(* CODESYS project p7lib-basetypes.library
   Company: MacGregor
   DocFormat: reStructuredText
   DefaultNamespace: p7type
   Version: 1.2.7
   Placeholder: p7lib-basetypes
   Author: Ralph Koettlitz
   Title: p7lib-basetypes

Project tree, tasks and I/O mapping:
  AnalogOut/
    interface IAnalogOut: Value
  Common/
    interface IAMSADDR: AMSAddr
    interface IP6Identifier: ID, IDname
    interface IP6OpState: OpState
    interface IP6State: State
    data type P6IdName
    data type P6OpState
    data type P6State
  ControlUnits/
    data type ControlUnitStates
    interface IBaseControlUnit: ActionSignal, ActivateWinch, Alarm, AutoAvailable, AutoMode, Calibrate, CooperatingWinchIsRotating, Disable, InControl, IsInControlOf, JoystickInCentre, ManualTorqueRequested, ManualTorqueSignal, PotmeterRaw, PotmeterReference, ReleaseControl, RequestedWinchMode, SetSelectedWinch, StopWinch, TurtleMode, TurtleModeRequested, VelocityRaw, VelocityReference
    interface IFishpumpControl: Softstart, Speed, start, stop
    interface INethaulerControl: TiltIn, TiltOut
    interface ITrawlControlUnit: JoystickPORT, JoystickSTBD, PotentiometerPORT, PotentiometerSTBD, TDE, TensionMaster, TensionMaxRef, TorqueButtonPORT, TorqueButtonSTBD, VelocityMaster, VelocityMaxRef
  Electrical/
    Drive/
      data type ConfigDriveMux
      data type DriveCMD
      data type DriveGearSet
      data type DriveIInverterArray
      data type DriveIServiceArray
      data type DriveMuxAllocationData
      data type DriveMuxAllocationValue
      interface IDrive: getGearRatio, getInverterArray, getSpeed, getSpeedMax, getTorque, getTorqueMax, getTorqueRel, getTorqueRelMax, IDName, isActivationPossible, isAtZeroSpeed, OpState, setOperation, setProcessValues, State
      interface IDriveGearSet: setGearSet
      interface IDriveMux: acquire, areInvertersDeactivated, getActiveInverters, getAvailableInverters, getAverageMotorSpeed, getAverageTorqueRel, getInverter, getInverterInterface, getInvertersOwned, getMotorFactor, hasActiveInvertersMin, hasInvertersMin, isAllocationPossible, isAtZeroSpeed, isBusy, release, setInverterOperation, setMotors, setProcessValues, SplitMode, update, updateSpeedRef
    Inverter/
      interface IEncoder: changeDirectionRawValue, changeDirectionValue, DirectionValue, DirectionValueRaw, resetAll, Resolution, setValueTo, Value, ValueRaw
      interface IEncoderBlock: Length
      interface IInverter: AMSAddr, Event, EventId, getEncoder, getMotor, getOpTime, getPower, getSpeed, getTorqueRel, isAtZeroSpeed, OpState, resetOpTime, setMotor, setOperation, setProcessValues, State
      interface IMotor: Active, resetOpTime, Temperature
      data type InverterCMD
    PMS/
      data type AFE_CMD
      interface IAFE: ChargeOverload, Event, EventId, FieldbusProblem, getOpTime, ID, IDName, OpState, PassiveMode, Power, PowerRegen, setOperation, State
      interface IPMS: attachAFE, attachInverter, delAllAFE, delAllInverters, LimitPowerRegenUsage, LimitPowerUsage, PassiveMode, PowerRegenUsage, PowerUsage, StopPowerUsage
    Softstarter/
      interface ISoftstarter: Active, Enabled, Error, Local, OpTime, PowerUsage, Ready, reset, Running, start, stop
  EStop/
    interface IEmergencyStop: Activated, ActivatedSwitchIdx, ActivatedSwitchName
  Events/
    Alarm Class Definitions.txt
    Alarm Definitions.txt
    data type EventIdentifier
    data type UnitTypeID
  00000000-0000-0000-0000-000000000000|Events\Alarm Class Definitions.txt
  00000000-0000-0000-0000-000000000000|Events\Alarm Definitions.txt
  Hydraulics/
    HPU/
      interface IHPUBrake: Active, Error, PressureOK, setActive
    Valve/
      interface IValve: CalibrationMode, Error, setValve
      data type ValveCMD
  NtoMProtocol/
    interface IProtoBase1ToN: attach, getNoServices, getServiceByIdx, isAttached, resetService
    interface IProtoBaseNTo1: attach, getMasterByIdx, getNoMasters, isAttached, resetServices
    interface IProtocol
    interface IProtoMasterSingleService: attach, getService
    interface IProtoService
  PID/
    data type ConfigPID
    data type ConfigPID2P
    data type ConfigTrawlController
    interface IPID2DController: Error, Out, update
    interface IPIDController: Error, Out, update
  Sensor/
    interface IAnalogSensor: Error
    interface IAnalogSensorBase: Value, ValueRaw
  Winch/
    data type ClutchCMD
    data type ClutchStates
    data type FreeWheelingBrakeStates
    data type FreeWheelingBrakeUserCMD
    interface IAnchorWinch
    interface IBaseUserWinch: AssignControlUnitInControl, AutoMode, BoostAllowed, ControlCanBeReleased, getVelocityReference, ID, IsReadyToActivate, IsRotating, Length, ManMode, SafetyDistance, SetLengthNull, Speed, SpeedMax, State, Tension, Torque, TorqueMax, TorqueRel, Velocity, winchDriverStopped
    interface IClutch: ClutchState, ParkingBrakesOnWhileJoystickInCenterEnabled, SetClutchOperation
    interface IClutchAndBrake: BrakeOffPressure, BrakeOnPressure, ClutchState, FreeWheelingBrakeState, ParkingBrakesOnWhileJoystickInCenterEnabled, SetClutchOperation, SetFreeWheelingBrakeOperation
    interface IFishpump: DifferentialPressure, EnvironmentalPressure, MotorhousePressure, OilTemperature, PressureLow, TemperatureHigh
    interface INetHaulerWinch: TiltIn, TiltOut
    interface ISpool: confirmWirePosition, HeadPosition, Name, OpState, PIDError, setManualOperation, setOffsetDiamondScrew, setOperation, setSpoolEndPositionInner, setSpoolEndPositionOuter, Speed, State
    interface ITrawlModeController: HaulInModeAllowed, LengthDifference, LengthDifferenceMax, LengthDifferenceWarning, LengthMaster, LengthSetpoint, PayoutModeAllowed, SafetyLength, setOperation, setSounderDifferenceToZero, SnagControl, SounderLengthDifference, SounderLengthDifferenceMax, SounderLengthDifferenceWarning, TDE, TowingModeAllowed
    interface ITrawlWinch: AutoAvailable, AutoMode, Radius, SafetyDistance, setOperation, TorqueAuto, VelocityAuto
    interface IWinchMode: Mode
    data type ManualSpoolCMD
    data type SpoolCMD
    data type TrawlMaster
    data type TrawlWinchCMD
    data type UserWinchStates
    data type WinchAutoModes
    data type WinchManualModes
    data type WinchModes
  global variables CycleTimeConstants
  global variables Math
  global variables Parameters
*)

// Common/P6IdName
TYPE 
	P6IdName : STRING(32) := 'HAS NO NAME'; 
END_TYPE

// Common/P6OpState
{attribute 'qualified_only'}
{attribute 'strict'}
(*
State For Operations
====================

These values are giving an information whether a unit is running or not
*)
TYPE P6OpState :
(
	NOTAVAILABLE	:= -1,
	STOPPED			:= 0,
	PAUSING			:= 1,
	PREPARE			:= 2,
	RUN  			:= 3
);
END_TYPE

// Common/P6State
{attribute 'qualified_only'}
{attribute 'strict'}
(*
Device State
============

These states are similar to the Ethercat statemachine. Don't confuse these states with
states for operation
*)
TYPE P6State :
(
	BUSY 		:= -1,			// no access because of concurrent operation
	INIT 		:= 0,			// Initializing objects
	PREOP 		:= 1,			// Check whether operation is possible
	OP			:= 2			// Full operational
) INT;
END_TYPE

// ControlUnits/ControlUnitStates
// The different states a control unit can be in.
{attribute 'qualified_only'}
{attribute 'strict'}
TYPE ControlUnitStates :
(
	INIT 		:= 0,
	MONITORING 	:= 1,
	REQ_CONTROL := 2,
	IN_CONTROL 	:= 3,
	CALIBRATE 	:= 4,
	PAYOUT		:= 5,
	HAULIN		:= 6,
	TOW			:= 7
);
END_TYPE

// Electrical/Drive/ConfigDriveMux
TYPE ConfigDriveMux :
	STRUCT
		ID						: DINT				:= -666;
		name					: P6IdName			:= '';
		contextChangeTimeMax	: TIME 				:= T#5S;
		contextChangeTimeMin	: TIME				:= T#1S;
	END_STRUCT
END_TYPE

// Electrical/Drive/DriveCMD
{attribute 'qualified_only'}
{attribute 'strict'}
TYPE DriveCMD:
(
	NONE 		:= 0,
	ACTIVATE 	:= 1, 	// Go to run state, magnetized and no motor change. 
	PAUSE 		:= 2,
	STOP 		:= 3, 	// Stop motor connected to inverter.
	RESET 		:= 4, 	// Reset inverter faults.
	FASTSTOP	:= 5
) INT;
END_TYPE

// Electrical/Drive/DriveGearSet
{attribute 'qualified_only'}
{attribute 'strict'}
TYPE DriveGearSet :
(
	DEFAULT := 0,
	SET2	:= 1
) DINT;
END_TYPE

// Electrical/Drive/DriveIInverterArray
// Array for inverters per drive
TYPE DriveIInverterArray : ARRAY[0..Parameters.InverterPoolSize-1] OF IInverter; END_TYPE

// Electrical/Drive/DriveIServiceArray
// Muxer Inverter Array
TYPE DriveIServiceArray : ARRAY[0..Parameters.MuxerInverterPoolSize-1] OF IProtoService; END_TYPE

// Electrical/Drive/DriveMuxAllocationData
(*
This type is used to configure allocation priority values in ConfigInverter. 
*) 
TYPE 
	DriveMuxAllocationData : 
		ARRAY[0..Parameters.MuxerInverterPoolSize-1] OF DriveMuxAllocationValue := 
			[Parameters.MuxerInverterPoolSize(DriveMuxAllocationValue.LVL_NIL)]; 
END_TYPE

// Electrical/Drive/DriveMuxAllocationValue
{attribute 'qualified_only'}
TYPE DriveMuxAllocationValue :
(
	LVL_NIL 	:= -1,
	LVL_1		:= 0,
	LVL_2		:= 1,
	LVL_3		:= 2,
	LVL_4		:= 3,
	LVL_NO_SW	:= 100
) DINT;
END_TYPE

// Electrical/Inverter/InverterCMD
{attribute 'qualified_only'}
{attribute 'strict'}
TYPE InverterCMD:
(
	NONE 		:= 0,
	ACTIVATE 	:= 1, 	// Go to run state, magnetized and no motor change. 
	PAUSE 		:= 2,
	STOP 		:= 3, 	// Stop motor connected to inverter.
	RESET 		:= 4 	// Reset inverter faults.
) INT;
END_TYPE

// Electrical/PMS/AFE_CMD
{attribute 'qualified_only'}
{attribute 'strict'}
TYPE AFE_CMD:
(
	NONE 		:= 0,
	RUN			:= 1, 
	STOP 		:= 3, 	// Stop motor connected to inverter.
	RESET 		:= 4 	// Reset inverter faults.
) INT;
END_TYPE

// Events/EventIdentifier
{attribute 'qualified_only'}
{attribute 'strict'}
TYPE EventIdentifier :
	(	
		NO_ERROR 														:= 16#00000000,
		
		// Inverters
		INVERTER_NO_POWER_SUPPLY										:= 16#00000001, // No power supply for the motor
		INVERTER_OVERVOLTAGE 											:= 16#00000002, // Inverter is indicating too much voltage 
		INVERTER_TRIPPED 												:= 16#00000003, // Inverter is indicating error
		INVERTER_COMM_FAULT 											:= 16#00000004, // Fieldbus problem
		INVERTER_WRONG_MOTOR	 										:= 16#00000005,	// Invalid motor number
		INVERTER_LOCAL 													:= 16#00000006, // Inverter is in local mode
		INV_NO_READYREF		 											:= 16#00000007, // Inverter doesn't build magnet field 
		INVERTER_NO_CONTACTOR_MSG 										:= 16#00000008, // Contactor signal indicates wrong state
		INVERTER_RESET_REQUEST 											:= 16#00000009,		
		INVERTER_NO_DC													:= 16#0000000A, // Frontend doesn't deliver DC
		
		// Drives
		DRIVE_NOT_ENOUGH_MOTORS 										:= 16#00000010, // When the number of motors is too low
		DRIVE_ACTIVATION_FAILED 										:= 16#00000011, // When an inverter couldn't be activated.
		DRIVE_NO_ENCODERS_AVAILABLE										:= 16#00000012, // Encoder isn't working 
		DRIVE_DIRECT_ENCODER_CHOICE_WRONG								:= 16#00000013,	// config.Option_OnlyThisInverterHasEncoder >= NumberOfInvertersMax	 

		// Winch Base 
		WINCHBASE_AUTOMODE_LARGELAG										:= 16#00000020,	// Too large lag between setpoint and length
		WINCHBASE_DRIVE_IS_NOT_AVAILABLE								:= 16#00000021,
		WINCHBASE_SPOOL_IS_NOT_AVAILABLE								:= 16#00000022, // The drive for spooling is down
	 
		// Encoder
		ENCODER_COUNTER_JITTER											:= 16#00000030,  // The counter is changing too fast
		
		// Spool
		SPOOL_CONFIG_ERROR												:= 16#00000040,	// Spool Drive Configuration error
		SPOOL_NO_DRIVE													:= 16#00000041, // Drive is missing
		
		// Motor Multiplexer											
		MMUX_SWITCHING_MOTOR											:= 16#00000050, // One of the inverters is controlling the wrong motor
		
		// AFE
		AFE_NO_NET														:= 16#00000060, // No net
		AFE_STARTUP_FAILED												:= 16#00000061,
		AFE_TRIPPED 													:= 16#00000062, // Inverter is indicating error
		AFE_COMM_FAULT 													:= 16#00000063, // Fieldbus problem
		AFE_LOCAL 														:= 16#00000064, // Inverter is in local mode
		AFE_RESET_REQUEST 												:= 16#00000065,		
		AFE_ESTOP		 												:= 16#00000066	
		
	) UDINT;
END_TYPE

// Events/UnitTypeID
{attribute 'qualified_only'}
{attribute 'strict'}
TYPE UnitTypeID :
(
	SYSTEM 								:= 16#00,
	CONFIG								:= 16#01,
	PMS									:= 16#02,
	HPU									:= 16#03,
	SENSOR								:= 16#04,
	INVERTER 							:= 16#05,
	SOFTSTARTER							:= 16#06,
	DRIVE 								:= 16#07,
	EWINCH								:= 16#08,
	WINCH	 							:= 16#09,
	PANEL								:= 16#0A,
	SPOOL								:= 16#1B,
	FISHPUMP							:= 16#1C,
	COOLING								:= 16#1D
) UDINT;
END_TYPE

// Hydraulics/Valve/ValveCMD
{attribute 'qualified_only'}
{attribute 'strict'}
TYPE ValveCMD :
(
	NONE		:= -1,
	OFF 		:= 0,
	ON 			:= 1,
	CALIBRATE	:= 2,
	RESET		:= 3
) DINT;
END_TYPE

// PID/ConfigPID
TYPE ConfigPID :
	STRUCT
		Kp : LREAL := 1.0;			// Gain
		Ki : LREAL := 0.0;			// Integration factor
		Kd : LREAL := 0.0;			// Differential gain
		Kf1 : LREAL := 0.0; 			// Feedforward gain 1 used by FFPid FB
		Kf2 : LREAL := 0.0; 			// Feedforward gain 2 used by FFPid FB
		Deadband : LREAL := 0.0;
		InitializeIntegrator : BOOL := FALSE; 
		IntegratorInit : LREAL := 0.0; 	// Integrator initial value 0..1 (aka %/100) of the output range/2
		Tau : LREAL := 1.0; 			// Filtering incomming values in %. 0.1 is 10% if a new value is used 
		NullValue : LREAL := 0.0;		// Output when the PID controller is deactivated
	END_STRUCT
END_TYPE

// PID/ConfigPID2P
(* 
Purpose
=======
This is a second parameter set for PID controllers where different directions
shall have different properties.

The first parameterset is for positive errors and the second is for negative errors.
All elements here are part of the second parameter set
*)
TYPE ConfigPID2P EXTENDS ConfigPID :
	STRUCT
		Kp2 	: LREAL := 1.0;			// Gain 2nd parametert set
		Ki2 	: LREAL := 0.0;			// Integration factor 2nd parametert set
		Kd2 	: LREAL := 0.0;			// Differential gain 2nd parametert set
		Kf12	: LREAL := 0.0;
		Kf22	: LREAL := 0.0;		
	END_STRUCT
END_TYPE

// PID/ConfigTrawlController
TYPE ConfigTrawlController :
	STRUCT
		KpVelocity					: LREAL := 0.02; 
		KpTorque					: LREAL := 0.0001;
		KiTorque					: LREAL := 0.001;
		KiVelocityLimit				: LREAL := 0.001;
		KiTensionLimit				: LREAL := 0.001;
		deadbandLength				: LREAL := 3.0;
	END_STRUCT
END_TYPE

// Winch/ClutchCMD
{attribute 'qualified_only'}
{attribute 'strict'}
TYPE ClutchCMD :
(
	NONE	:= 0,
	Engage := 1,
	DisEngage := 2
);
END_TYPE

// Winch/ClutchStates
{attribute 'qualified_only'}
{attribute 'strict'}
TYPE ClutchStates :
(
	Initialize 			:= 0,		// Clutch is initializing
	DisengageStartup	:= 1,
	DisengageRun		:= 2,
	Disengaged			:= 3,
	EngageStartup		:= 4,
	EngageWait			:= 5,
	EngageRun			:= 6,
	Engaged				:= 7,	
	Idle				:= 8,
	Error 				:= 99		// Clutch is in error position => both engaged and disengaged sensor is activated
);
END_TYPE

// Winch/FreeWheelingBrakeStates
{attribute 'qualified_only'}
{attribute 'strict'}
TYPE FreeWheelingBrakeStates :
(
	BrakeControlDisabled := 0,				// Brakes are controlled by winch/clutch
	BrakeControlEnabled := 1				// Brakes are controlled by potmeter on control unit in control					
);
END_TYPE

// Winch/FreeWheelingBrakeUserCMD
// CMD from user control
{attribute 'qualified_only'}
{attribute 'strict'}
TYPE FreeWheelingBrakeUserCMD :
(
	DisableBrakeControl := 0,				// Brakes are controlled by winch/clutch
	EnableBrakeControl := 1					// Brakes are controlled by potmeter on control unit in control	
);
END_TYPE

// Winch/ManualSpoolCMD
{attribute 'qualified_only'}
{attribute 'strict'}
TYPE ManualSpoolCMD :
(
	STOP := 0,
	TOSTART := 1,
	TOEND := 2
) DINT;
END_TYPE

// Winch/SpoolCMD
{attribute 'qualified_only'}
{attribute 'strict'}
TYPE SpoolCMD :
	(
		NONE 		:= 0,
		AUTO		:= 1,
		PAUSE		:= 2,
		STOP		:= 3,
		OFF			:= 4,
		MANUAL		:= 5,
		CALIBRATE	:= 6,
		RESET		:= 7,
		FASTSTOP	:= 8
	) DINT;
END_TYPE

// Winch/TrawlMaster
{attribute 'qualified_only'}
{attribute 'strict'}
TYPE TrawlMaster :
(
	AVERAGE		:= 0,
	STBD 		:= 1,
	PORT		:= 2,
	MID			:= 3,
	RUDDER		:= 5,
	SHORTEST	:= 6,
	LONGEST		:= 7 
) DINT;
END_TYPE

// Winch/TrawlWinchCMD
{attribute 'qualified_only'}
{attribute 'strict'}
TYPE TrawlWinchCMD :
(
	NONE							:= 0,
	STOP							:= 1,
	MANUAL_MODE						:= 2,
	TOWING							:= 3,			
	HAULIN_TO_SETPOINT				:= 4,
	HAULIN_TO_SAFETY_RANGE			:= 5,
	PAYOUT_TO_SETPOINT				:= 6	
) DINT;
END_TYPE

// Winch/UserWinchStates
{attribute 'qualified_only'}
{attribute 'strict'}
TYPE UserWinchStates :
(
	INACTIVE 				:= 0,			// winch is inactive

	MANUAL					:= 100,
	MANUAL_PREPARE			:= 101,			// Winch sends commands to EWinch to start
	MANUAL_PREPARE2			:= 102,			// Winch sends commands to EWinch to start
	MANUAL_PREOP			:= 103,			// Winch is waiting for EWinch to go out of prepare
	MANUAL_ACTIVE			:= 104,			// Winch is running ok
	MANUAL_ACTIVE_REDUCED	:= 105,

	CONST_TORQUE			:= 200,
	CONST_TORQUE_PREPARE	:= 201,			// Winch sends commands to EWinch to start
	CONST_TORQUE_PREPARE2	:= 202,			// Winch sends commands to EWinch to start
	CONST_TORQUE_PREOP		:= 203,			// Winch is waiting for EWinch to go out of prepare
	CONST_TORQUE_ACTIVE		:= 204,			// Winch is running ok	
	
	AUTO					:= 300,
	AUTO_PREPARE			:= 301,
	AUTO_PREPARE2			:= 302,
	AUTO_PREOP				:= 303,
	AUTO_ACTIVE				:= 304,
	
	PAYOUT_TRAWL			:= 400,
	PAYOUT_TRAWL_PREPARE	:= 401,
	PAYOUT_TRAWL_PREOP		:= 402,
	PAYOUT_TRAWL_ACTIVE		:= 403,

	HAULIN_TRAWL			:= 500,
	HAULIN_TRAWL_PREPARE	:= 501,
	HAULIN_TRAWL_PREOP		:= 502,
	HAULIN_TRAWL_ACTIVE		:= 503,
	
	TOWING					:= 600,
	TOWING_PREPARE			:= 601,
	TOWING_PREOP			:= 602,
	TOWING_ACTIVE			:= 603,
	
	SLAVE					:= 700,
	SLAVE_PREPARE			:= 701,
	SLAVE_PREOP				:= 702,
	SLAVEACTIVE				:= 703,
	
	EMERGENCYSTOP 			:= 1000
) DINT;
END_TYPE

// Winch/WinchAutoModes
{attribute 'qualified_only'}
{attribute 'strict'}
TYPE WinchAutoModes :
(
	MANUAL 			:= 0,
	AUTO 			:= 1,
	PAYOUT_TRAWL	:= 2,
	HAULIN_TRAWL	:= 3,
	TOWING_TRAWL	:= 4
);
END_TYPE

// Winch/WinchManualModes
{attribute 'qualified_only'}
{attribute 'strict'}
TYPE WinchManualModes :
	(
		NORMAL 				:= 0,
		MANUAL_TORQUE 		:= 1,
		CONSTANT_TORQUE 	:= 2,
		TWO_SPEED 			:= 3,
		BOOST 				:= 4
	) DINT;
END_TYPE

// Winch/WinchModes
(*
	This is for the mode of a BaseUserWinch

*)
{attribute 'qualified_only'}
{attribute 'strict'}
TYPE WinchModes :
(
	ESTOP			:= -1,
	IDLE 			:= 0,
	MANUAL			:= 1,
	PAYOUT			:= 2,
	HAULIN			:= 3,
	AUTO			:= 4,
	TRAWL			:= 5,
	TORQUE			:= 6,
	SLAVE			:= 7
) DINT;
END_TYPE

// CycleTimeConstants
(*
This cyle time constants are used for PID controllers and trajectory generators.
The constants are organized like layers. 
*)
VAR_GLOBAL CONSTANT
	CycleTime_Task0 : TIME := T#10MS; 	// The time for the cycle time of a task	
	CycleTime_Task1 : TIME := T#10MS; 	// The time for the cycle time of a task	
	CycleTime_Task2 : TIME := T#10MS; 	// The time for the cycle time of a task	
	CycleTime_Task3 : TIME := T#10MS; 	// The time for the cycle time of a task

	CycleTime_PID0	: TIME := T#50MS; 	// Cycle time for PID controllers. 
										// A inverter delivers data every 20ms
										// which makes this to a save choice		
	CycleTime_PID1	: TIME := T#200MS; 	// Cycle time for PID controllers. 
	CycleTime_PID2	: TIME := T#400MS; 	// Cycle time for PID controllers. 
END_VAR

// Math
{attribute 'qualified_only'}
VAR_GLOBAL CONSTANT
	PI 					: LREAL := 3.141592653589793;
	PI2 				: LREAL := 6.283185307179586;
END_VAR

// Parameters
{attribute 'qualified_only'}
VAR_GLOBAL CONSTANT
	// Size is always an array limit hence amount of elements minus 1
	inverterGroupSize		: DINT 		:= 100;
	MuxerInverterPoolSize	: DINT		:= 10;		// Inverters per pool of the muxer
	InverterPoolSize		: DINT		:= 8;		// Inverters per drive
	// Drives
	DriveArraySize			: DINT		:= 100;
	
END_VAR

// AnalogOut/IAnalogOut
INTERFACE IAnalogOut

{attribute 'monitoring' := 'call'}
{attribute 'TcRpcEnable'}
PROPERTY Value : LREAL
SET
END_SET
END_PROPERTY

END_INTERFACE

// Common/IAMSADDR
INTERFACE IAMSADDR

PROPERTY AMSAddr : AMSADDR
GET
END_GET
END_PROPERTY

END_INTERFACE

// Common/IP6Identifier
INTERFACE IP6Identifier

{attribute 'monitoring' := 'call'}
{attribute 'TcRpcEnable'}
PROPERTY ID : DINT
GET
END_GET
SET
END_SET
END_PROPERTY

{attribute 'monitoring' := 'call'}
{attribute 'TcRpcEnable'}
PROPERTY IDname : P6IdName
GET
END_GET
SET
END_SET
END_PROPERTY

END_INTERFACE

// Common/IP6OpState
INTERFACE IP6OpState

{attribute 'monitoring' := 'call'}
{attribute 'TcRpcEnable'}
PROPERTY OpState : P6OpState
GET
END_GET
END_PROPERTY

END_INTERFACE

// Common/IP6State
INTERFACE IP6State

{attribute 'monitoring' := 'call'}
{attribute 'TcRpcEnable'}
PROPERTY State : P6State
GET
END_GET
END_PROPERTY

END_INTERFACE

// ControlUnits/IBaseControlUnit
// Represents base interface for all control unit s.
INTERFACE IBaseControlUnit  EXTENDS __System.IQueryInterface

// When using MasterControl, this signal is used to activate other winches
{attribute 'monitoring':='call'}
{attribute 'TcRpcEnable'}
PROPERTY ActionSignal : BOOL
GET
END_GET
END_PROPERTY

{attribute 'monitoring':='call'}
{attribute 'TcRpcEnable'}
PROPERTY ActivateWinch : BOOL
GET
END_GET
END_PROPERTY

// If alarm in system call method with alarmState = TRUE
{attribute 'TcRpcEnable'}
METHOD Alarm : BOOL
VAR_INPUT
	alarmState : BOOL;
END_VAR
END_METHOD

PROPERTY AutoAvailable : BOOL
GET
END_GET
END_PROPERTY

PROPERTY AutoMode : BOOL
SET
END_SET
END_PROPERTY

{attribute 'monitoring':='call'}
{attribute 'TcRpcEnable'}
METHOD Calibrate : BOOL
END_METHOD

// When using MasterControl, this indicates that the cooperating winch is rotating so that this winch cant timeout. 
{attribute 'monitoring':='call'}
{attribute 'TcRpcEnable'}
PROPERTY CooperatingWinchIsRotating : BOOL
GET
END_GET
END_PROPERTY

PROPERTY Disable : BOOL
SET
END_SET
END_PROPERTY

{attribute 'monitoring':='call'}
{attribute 'TcRpcEnable'}
PROPERTY InControl : BOOL
GET
END_GET
END_PROPERTY

// Returns TRUE if the control unit is in control of the winch with winchID
{attribute 'TcRpcEnable'}
METHOD IsInControlOf : BOOL
VAR_INPUT
	winchID : DINT;
END_VAR
END_METHOD

{attribute 'monitoring':='call'}
{attribute 'TcRpcEnable'}
PROPERTY JoystickInCentre : BOOL
GET
END_GET
END_PROPERTY

// When using MasterControl, this signal is used to activate manual torque on other winches
{attribute 'monitoring':='call'}
{attribute 'TcRpcEnable'}
PROPERTY ManualTorqueRequested : BOOL
GET
END_GET
END_PROPERTY

{attribute 'monitoring':='call'}
{attribute 'TcRpcEnable'}
// Read true when man torque is pressed
 PROPERTY ManualTorqueSignal : BOOL
GET
END_GET
END_PROPERTY

{attribute 'monitoring':='call'}
{attribute 'TcRpcEnable'}
PROPERTY PotmeterRaw : LREAL
GET
END_GET
END_PROPERTY

// The actual potmeter value used by winch
{attribute 'monitoring':='call'}
{attribute 'TcRpcEnable'}
PROPERTY PotmeterReference : LREAL
GET
END_GET
END_PROPERTY

{attribute 'TcRpcEnable'}
METHOD ReleaseControl : BOOL
VAR_INPUT
	winchID : DINT;
END_VAR
END_METHOD

{attribute 'monitoring':='call'}
{attribute 'TcRpcEnable'}
PROPERTY RequestedWinchMode : WinchManualModes
GET
END_GET
END_PROPERTY

{attribute 'TcRpcEnable'}
METHOD SetSelectedWinch : BOOL
VAR_INPUT
	winchToControl : IBaseUserWinch;
END_VAR
END_METHOD

{attribute 'monitoring':='call'}
{attribute 'TcRpcEnable'}
PROPERTY StopWinch : BOOL
GET
END_GET
SET
END_SET
END_PROPERTY

// TRUE if control unit requests turtle mode. Used by winch
{attribute 'monitoring':='call'}
{attribute 'TcRpcEnable'}
PROPERTY TurtleMode : BOOL
GET
END_GET
END_PROPERTY

// When using MasterControl, this signal is used to control turtle mode on other winches
{attribute 'monitoring':='call'}
{attribute 'TcRpcEnable'}
PROPERTY TurtleModeRequested : BOOL
GET
END_GET
END_PROPERTY

{attribute 'monitoring':='call'}
{attribute 'TcRpcEnable'}
PROPERTY VelocityRaw : LREAL
GET
END_GET
END_PROPERTY

// The value from control unit that controls the velocity of the winch
{attribute 'monitoring':='call'}
{attribute 'TcRpcEnable'}
PROPERTY VelocityReference : LREAL
GET
END_GET
END_PROPERTY

END_INTERFACE

// Winch/IBaseUserWinch
// Common winch interface used by control units etc.
INTERFACE IBaseUserWinch EXTENDS __SYSTEM.IQueryInterface, IP6OpState, IWinchMode

(* Assigns the control unit that is granted control bu ControlUnitMux to _controlUnitInControl *)
(*  __QUERYINTERFACE(controlUnitInControl, _controlUnitInControl) type converts from 	*)
(* IControlUnit to IStandardJoystickControlUnit to get velocity and torque values.		*)
(* If controlUnitInControl = 0, controlUnitInControl is unasigned						*)
{attribute 'TcRpcEnable'}
METHOD AssignControlUnitInControl : BOOL
VAR_INPUT
	controlUnitInControl : IBaseControlUnit;
END_VAR
END_METHOD

// Handshake between user control and winch
PROPERTY AutoMode : BOOL
SET
END_SET
END_PROPERTY

// True when winch is allowed to boost
{attribute 'monitoring':='call'}
{attribute 'TcRpcEnable'}
PROPERTY BoostAllowed : BOOL
GET
END_GET
END_PROPERTY

// Control of winch from control unit can be released. Means that winch is not moving, etc. 
{attribute 'TcRpcEnable'}
PROPERTY ControlCanBeReleased : BOOL
GET
END_GET
END_PROPERTY

{attribute 'TcRpcEnable'}
METHOD getVelocityReference : LREAL
END_METHOD

// The uniqe winch identificator
{attribute 'TcRpcEnable'}
PROPERTY ID : DINT
GET
END_GET
END_PROPERTY

// True when winch is ready to be activated
{attribute 'monitoring':='call'}
{attribute 'TcRpcEnable'}
PROPERTY IsReadyToActivate : BOOL
GET
END_GET
END_PROPERTY

(* When the winch is rotating faster than config.winchIsRotatingValue this property is true *)
{attribute 'monitoring':='call'}
{attribute 'TcRpcEnable'}
PROPERTY IsRotating : BOOL
GET
END_GET
END_PROPERTY

// Wire length in meters
{attribute 'monitoring':='call'}
{attribute 'TcRpcEnable'}
PROPERTY Length : LREAL
GET
END_GET
END_PROPERTY

// The current manual mode the winch is running in
{attribute 'TcRpcEnable'}
PROPERTY ManMode : WinchManualModes
GET
END_GET
END_PROPERTY

{attribute 'monitoring':='call'}
{attribute 'TcRpcEnable'}
PROPERTY SafetyDistance : LREAL
GET
END_GET
END_PROPERTY

// Resets length of wire to 0
{attribute 'TcRpcEnable'}
METHOD SetLengthNull : BOOL
END_METHOD

// Winch rotation speed in RPM
{attribute 'monitoring':='call'}
{attribute 'TcRpcEnable'}
PROPERTY Speed : LREAL
GET
END_GET
END_PROPERTY

// Maximum rotation speed in RPM for this winch
{attribute 'monitoring':='call'}
{attribute 'TcRpcEnable'}
PROPERTY SpeedMax : LREAL
GET
END_GET
END_PROPERTY

// The current state of the winch
{attribute 'TcRpcEnable'}
PROPERTY State : UserWinchStates
GET
END_GET
END_PROPERTY

// Wire tension in Kg
{attribute 'monitoring':='call'}
{attribute 'TcRpcEnable'}
PROPERTY Tension : LREAL
GET
END_GET
END_PROPERTY

// Wire torque in Nm
{attribute 'monitoring':='call'}
{attribute 'TcRpcEnable'}
PROPERTY Torque : LREAL
GET
END_GET
END_PROPERTY

// Maximum Wire torque in Nm for this winch
{attribute 'monitoring':='call'}
{attribute 'TcRpcEnable'}
PROPERTY TorqueMax : LREAL
GET
END_GET
END_PROPERTY

// Wire torque in %, range 0-1
{attribute 'monitoring':='call'}
{attribute 'TcRpcEnable'}
PROPERTY TorqueRel : LREAL
GET
END_GET
END_PROPERTY

// Winch velocity in m/sec
{attribute 'monitoring':='call'}
{attribute 'TcRpcEnable'}
PROPERTY Velocity :  LREAL
GET
END_GET
END_PROPERTY

{attribute 'TcRpcEnable'}
METHOD winchDriverStopped : BOOL
END_METHOD

END_INTERFACE

// Winch/IWinchMode
INTERFACE IWinchMode

{attribute 'monitoring' := 'call'}
(* This is the unified state of the state of operation *)
{attribute 'TcRpcEnable'}
PROPERTY Mode : WinchModes
GET
END_GET
END_PROPERTY

END_INTERFACE

// ControlUnits/IFishpumpControl
INTERFACE IFishpumpControl EXTENDS IBaseControlUnit

{attribute 'monitoring':='call'}
{attribute 'TcRpcEnable'}
PROPERTY Softstart : BOOL
GET
END_GET
SET
END_SET
END_PROPERTY

{attribute 'monitoring':='call'}
{attribute 'TcRpcEnable'}
PROPERTY Speed : LREAL
GET
END_GET
SET
END_SET
END_PROPERTY

{attribute 'TcRpcEnable'}
METHOD start : BOOL
END_METHOD

{attribute 'TcRpcEnable'}
METHOD stop : BOOL
END_METHOD

END_INTERFACE

// ControlUnits/INethaulerControl
INTERFACE INethaulerControl

PROPERTY TiltIn : BOOL
GET
END_GET
END_PROPERTY

PROPERTY TiltOut : BOOL
GET
END_GET
END_PROPERTY

END_INTERFACE

// ControlUnits/ITrawlControlUnit
INTERFACE ITrawlControlUnit EXTENDS IBaseControlUnit

// TRUE if joystick axis in centre
{attribute 'monitoring':='call'}
{attribute 'TcRpcEnable'}
PROPERTY JoystickPORT : LREAL
GET
END_GET
END_PROPERTY

// TRUE if joystick axis in centre
{attribute 'monitoring':='call'}
{attribute 'TcRpcEnable'}
PROPERTY JoystickSTBD : LREAL
GET
END_GET
END_PROPERTY

// TRUE if joystick axis in centre
{attribute 'monitoring':='call'}
{attribute 'TcRpcEnable'}
PROPERTY PotentiometerPORT : LREAL
GET
END_GET
END_PROPERTY

// TRUE if joystick axis in centre
{attribute 'monitoring':='call'}
{attribute 'TcRpcEnable'}
PROPERTY PotentiometerSTBD : LREAL
GET
END_GET
END_PROPERTY

{attribute 'TcRpcEnable'}
{attribute 'monitoring':='call'}
PROPERTY TDE : BOOL
GET
END_GET
SET
END_SET
END_PROPERTY

{attribute 'TcRpcEnable'}
{attribute 'monitoring':='call'}
PROPERTY TensionMaster : LREAL
GET
END_GET
END_PROPERTY

{attribute 'TcRpcEnable'}
{attribute 'monitoring':='call'}
PROPERTY TensionMaxRef : LREAL
GET
END_GET
SET
END_SET
END_PROPERTY

// TRUE if joystick axis in centre
{attribute 'monitoring':='call'}
{attribute 'TcRpcEnable'}
PROPERTY TorqueButtonPORT : BOOL
GET
END_GET
END_PROPERTY

// TRUE if joystick axis in centre
{attribute 'monitoring':='call'}
{attribute 'TcRpcEnable'}
PROPERTY TorqueButtonSTBD : BOOL;
GET
END_GET
END_PROPERTY

{attribute 'TcRpcEnable'}
{attribute 'monitoring':='call'}
PROPERTY VelocityMaster : LREAL
GET
END_GET
END_PROPERTY

{attribute 'TcRpcEnable'}
{attribute 'monitoring':='call'}
PROPERTY VelocityMaxRef : LREAL
GET
END_GET
SET
END_SET
END_PROPERTY

END_INTERFACE

// Electrical/Drive/IDrive
INTERFACE IDrive EXTENDS IP6Identifier, IP6OpState, IProtoBase1ToN, IDriveGearSet

METHOD getGearRatio : LREAL
END_METHOD

{attribute 'TcRpcEnable'}
METHOD getInverterArray : REFERENCE TO DriveIInverterArray
END_METHOD

{attribute 'TcRpcEnable'}
METHOD getSpeed : LREAL
END_METHOD

{attribute 'TcRpcEnable'}
METHOD getSpeedMax : LREAL
END_METHOD

{attribute 'TcRpcEnable'}
METHOD getTorque : LREAL
END_METHOD

{attribute 'TcRpcEnable'}
METHOD getTorqueMax : LREAL
END_METHOD

{attribute 'TcRpcEnable'}
METHOD getTorqueRel : LREAL
END_METHOD

{attribute 'TcRpcEnable'}
METHOD getTorqueRelMax : LREAL
END_METHOD

{attribute 'monitoring' := 'call'}
{attribute 'TcRpcEnable'}
PROPERTY IDName : P6IdName
GET
END_GET
END_PROPERTY

{attribute 'TcRpcEnable'}
METHOD isActivationPossible : BOOL
END_METHOD

{attribute 'TcRpcEnable'}
METHOD isAtZeroSpeed : BOOL
END_METHOD

{attribute 'monitoring' := 'call'}
{attribute 'TcRpcEnable'}
PROPERTY OpState : P6OpState
GET
END_GET
END_PROPERTY

{attribute 'TcRpcEnable'}
METHOD setOperation : BOOL
VAR_INPUT
	CMD : DriveCMD;
END_VAR
END_METHOD

{attribute 'TcRpcEnable'}
METHOD PUBLIC setProcessValues : BOOL
VAR_INPUT
	Speed : LREAL;
	TorqueRel : LREAL;
END_VAR
END_METHOD

{attribute 'monitoring' := 'call'}
{attribute 'TcRpcEnable'}
PROPERTY State : P6State
GET
END_GET
END_PROPERTY

END_INTERFACE

// NtoMProtocol/IProtoBase1ToN
INTERFACE IProtoBase1ToN EXTENDS IProtocol

{attribute 'monitoring' := 'call'}
METHOD attach : IProtoBase1ToN
VAR_INPUT
	Service : IProtoService;
END_VAR
END_METHOD

{attribute 'monitoring' := 'call'}
METHOD getNoServices : DINT
END_METHOD

{attribute 'monitoring' := 'call'}
METHOD getServiceByIdx : IProtoService
VAR_INPUT
	Index  : DINT;
END_VAR
END_METHOD

{attribute 'monitoring' := 'call'}
METHOD isAttached : BOOL
VAR_INPUT
	Service : IProtoService;
END_VAR
END_METHOD

{attribute 'monitoring' := 'call'}
METHOD resetService : IProtoBase1ToN
END_METHOD

END_INTERFACE

// NtoMProtocol/IProtocol
(*
	This is the foundation of all protocols
*)
INTERFACE IProtocol EXTENDS __SYSTEM.IQueryInterface

END_INTERFACE

// NtoMProtocol/IProtoService
(*
This interface defines a simple service, used when the service
is the passive part of getting attached
*)
INTERFACE IProtoService EXTENDS IProtocol

END_INTERFACE

// Electrical/Drive/IDriveGearSet
INTERFACE IDriveGearSet

METHOD setGearSet : BOOL  
VAR_INPUT
	GearSet : DriveGearSet ;
END_VAR
END_METHOD

END_INTERFACE

// Electrical/Drive/IDriveMux
INTERFACE IDriveMux EXTENDS IP6Identifier, IProtoBase1ToN

METHOD acquire : BOOL
VAR_INPUT
	ID 					: DINT; 
	Motor				: DINT;
	MotorQuantitySTD 	: DINT; 
	MotorQuantitySPM 	: DINT; 	
	OptionMotorSnatch	: BOOL;
	Data				: REFERENCE TO DriveMuxAllocationData;
END_VAR
END_METHOD

METHOD areInvertersDeactivated : BOOL
VAR_INPUT
	ID		: DINT;
END_VAR
END_METHOD

METHOD getActiveInverters : DINT
VAR_INPUT
	ID : DINT;
END_VAR
END_METHOD

METHOD getAvailableInverters : DINT
VAR_INPUT
	ID : DINT;
END_VAR
END_METHOD

METHOD getAverageMotorSpeed : LREAL
VAR_INPUT
	ID : DINT;
END_VAR
END_METHOD

METHOD getAverageTorqueRel : LREAL
VAR_INPUT
	ID : DINT;
END_VAR
END_METHOD

METHOD getInverter : IInverter
VAR_INPUT
	ID		: DINT;
	Index	: DINT;
END_VAR
END_METHOD

METHOD getInverterInterface : IInverter
VAR_INPUT
	Index : DINT;
END_VAR
END_METHOD

METHOD getInvertersOwned : DINT
VAR_INPUT
	ID : DINT;
END_VAR
END_METHOD

METHOD getMotorFactor : LREAL
VAR_INPUT
	ID				: DINT;
	AllocationData	: REFERENCE TO DriveMuxAllocationData;	
END_VAR
END_METHOD

METHOD hasActiveInvertersMin : BOOL
VAR_INPUT
	ID : DINT;
END_VAR
END_METHOD

METHOD hasInvertersMin : BOOL
VAR_INPUT
	ID : DINT;
END_VAR
END_METHOD

(*
	IsAllocationPossible 
	
	Return Value: Boolean for success
	
	This method is indicating success when enough inverters can be allocated, which includes
	they have to be in state OP
*)
METHOD isAllocationPossible : BOOL
VAR_INPUT
	ID 							: DINT; 
	Motor						: DINT;
	MotorQuantitySTD 			: DINT; 	
	MotorQuantitySPM 			: DINT; 	
	OptionMotorCanBeSnatched 	: BOOL;
END_VAR
VAR_INPUT CONSTANT
	Data						: REFERENCE TO DriveMuxAllocationData;	
END_VAR
END_METHOD

METHOD isAtZeroSpeed : BOOL
VAR_INPUT
	ID : DINT;
END_VAR
END_METHOD

METHOD isBusy : BOOL
VAR_INPUT
	ID		: DINT;
END_VAR
END_METHOD

METHOD release : BOOL
VAR_INPUT
	ID : DINT;
END_VAR
END_METHOD

METHOD setInverterOperation : BOOL
VAR_INPUT
	ID : DINT;
	CMD : InverterCMD;
END_VAR
END_METHOD

METHOD setMotors : BOOL
VAR_INPUT
	ID 			: DINT;
END_VAR
END_METHOD

METHOD setProcessValues : BOOL
VAR_INPUT
	ID 			: DINT;
	Speed 		: LREAL;
	TorqueRel	: LREAL;
END_VAR
END_METHOD

{attribute 'TcRpcEnable'}
PROPERTY SplitMode : BOOL
GET
END_GET
SET
END_SET
END_PROPERTY

METHOD update : BOOL
VAR_INPUT
	Config 							: REFERENCE TO ConfigDriveMux;
END_VAR
END_METHOD

METHOD updateSpeedRef : BOOL
VAR_INPUT
	ID 			: DINT;
	SpeedRef	: LREAL;
END_VAR
END_METHOD

END_INTERFACE

// Electrical/Inverter/IInverter
INTERFACE IInverter EXTENDS IP6Identifier, 
							IP6State, 
							IP6OpState, 
							IProtoService, 
							IAMSADDR

(*
Purpose
=======
This interface provides a property promise to access the AMSADDR of a Twincat System

*)
{attribute 'TcRpcEnable'}
PROPERTY AMSAddr : AMSADDR
GET
END_GET
END_PROPERTY

{attribute 'monitoring' := 'call'}
{attribute 'TcRpcEnable'}
PROPERTY Event : BOOL
GET
END_GET
END_PROPERTY

{attribute 'monitoring' := 'call'}
{attribute 'TcRpcEnable'}
PROPERTY EventId : EventIdentifier
GET
END_GET
END_PROPERTY

{attribute 'TcRpcEnable'}
METHOD getEncoder : IEncoder
VAR_INPUT
	Index	: UDINT;
END_VAR
END_METHOD

{attribute 'TcRpcEnable'}
METHOD getMotor : DINT
END_METHOD

{attribute 'monitoring' := 'call'}
{attribute 'TcRpcEnable'}
METHOD getOpTime : TIME
VAR_INPUT
	Index : DINT;
END_VAR
END_METHOD

{attribute 'monitoring' := 'call'}
{attribute 'TcRpcEnable'}
METHOD getPower : LREAL
END_METHOD

{attribute 'TcRpcEnable'}
{attribute 'monitoring' := 'call'}
METHOD getSpeed : LREAL
END_METHOD

{attribute 'TcRpcEnable'}
{attribute 'monitoring' := 'call'}
METHOD getTorqueRel : LREAL
END_METHOD

{attribute 'TcRpcEnable'}
METHOD isAtZeroSpeed : BOOL
END_METHOD

{attribute 'monitoring' := 'call'}
{attribute 'TcRpcEnable'}
PROPERTY OpState : P6OpState
GET
END_GET
END_PROPERTY

{attribute 'TcRpcEnable'}
METHOD resetOpTime : BOOL
END_METHOD

{attribute 'TcRpcEnable'}
METHOD setMotor : BOOL
VAR_INPUT
	Index : DINT;
END_VAR
END_METHOD

{attribute 'TcRpcEnable'}
METHOD setOperation : BOOL
VAR_INPUT
	Operation	: InverterCMD;
END_VAR
END_METHOD

{attribute 'TcRpcEnable'}
METHOD setProcessValues : BOOL
VAR_INPUT
	Speed	: LREAL;
	TorqueRel	: LREAL;
END_VAR
END_METHOD

{attribute 'monitoring' := 'call'}
{attribute 'TcRpcEnable'}
PROPERTY State : P6State
GET
END_GET
END_PROPERTY

END_INTERFACE

// Electrical/Inverter/IEncoder
INTERFACE IEncoder EXTENDS IProtoService

{attribute 'TcRpcEnable'}
METHOD changeDirectionRawValue : BOOL
END_METHOD

{attribute 'TcRpcEnable'}
METHOD changeDirectionValue : BOOL
END_METHOD

// Alternative to changeDirectionValue() call
{attribute 'TcRpcEnable'}
{attribute 'monitoring' := 'call'}
PROPERTY DirectionValue : BOOL
GET
END_GET
SET
END_SET
END_PROPERTY

// Alternative to changeDirectionValueRaw() call
{attribute 'TcRpcEnable'}
{attribute 'monitoring' := 'call'}
PROPERTY DirectionValueRaw : BOOL
GET
END_GET
SET
END_SET
END_PROPERTY

{attribute 'TcRpcEnable'}
METHOD resetAll : BOOL
END_METHOD

{attribute 'TcRpcEnable'}
{attribute 'monitoring' := 'call'}
PROPERTY Resolution : DINT
GET
END_GET
END_PROPERTY

{attribute 'TcRpcEnable'}
METHOD setValueTo : BOOL
VAR_INPUT
	NewValue : LINT;
END_VAR
END_METHOD

{attribute 'TcRpcEnable'}
{attribute 'monitoring' := 'call'}
PROPERTY Value : LINT
GET
END_GET
END_PROPERTY

{attribute 'TcRpcEnable'}
{attribute 'monitoring' := 'call'}
PROPERTY ValueRaw : LINT
GET
END_GET
END_PROPERTY

END_INTERFACE

// Electrical/Inverter/IEncoderBlock
INTERFACE IEncoderBlock EXTENDS IEncoder

{attribute 'TcRpcEnable'}
PROPERTY Length : LREAL
GET
END_GET
SET
END_SET
END_PROPERTY

END_INTERFACE

// Electrical/Inverter/IMotor
INTERFACE IMotor

{attribute 'monitoring' := 'call'}
{attribute 'TcRpcEnable'}
PROPERTY Active : BOOL
GET
END_GET
SET
END_SET
END_PROPERTY

{attribute 'TcRpcEnable'}
METHOD resetOpTime : BOOL
END_METHOD

{attribute 'monitoring' := 'call'}
{attribute 'TcRpcEnable'}
PROPERTY Temperature : LREAL
GET
END_GET
END_PROPERTY

END_INTERFACE

// Electrical/PMS/IAFE
INTERFACE IAFE EXTENDS IP6Identifier, IProtoBaseNTo1

{attribute 'monitoring' := 'call'}
{attribute 'TcRpcEnable'}
PROPERTY ChargeOverload : BOOL
GET
END_GET
END_PROPERTY

{attribute 'monitoring' := 'call'}
{attribute 'TcRpcEnable'}
PROPERTY Event : BOOL
GET
END_GET
END_PROPERTY

{attribute 'monitoring' := 'call'}
{attribute 'TcRpcEnable'}
PROPERTY EventId : EventIdentifier
GET
END_GET
END_PROPERTY

{attribute 'monitoring' := 'call'}
{attribute 'TcRpcEnable'}
PROPERTY FieldbusProblem : BOOL
GET
END_GET
END_PROPERTY

{attribute 'TcRpcEnable'}
METHOD getOpTime : TIME
END_METHOD

{attribute 'monitoring' := 'call'}
{attribute 'TcRpcEnable'}
PROPERTY ID : DINT
GET
END_GET
SET
END_SET
END_PROPERTY

{attribute 'monitoring' := 'call'}
{attribute 'TcRpcEnable'}
PROPERTY IDName : P6IdName
GET
END_GET
SET
END_SET
END_PROPERTY

{attribute 'monitoring' := 'call'}
{attribute 'TcRpcEnable'}
PROPERTY OpState : P6OpState
GET
END_GET
END_PROPERTY

{attribute 'monitoring' := 'call'}
{attribute 'TcRpcEnable'}
PROPERTY PassiveMode : BOOL
GET
END_GET
SET
END_SET
END_PROPERTY

{attribute 'monitoring' := 'call'}
{attribute 'TcRpcEnable'}
PROPERTY Power : LREAL
GET
END_GET
END_PROPERTY

{attribute 'monitoring' := 'call'}
{attribute 'TcRpcEnable'}
PROPERTY PowerRegen : LREAL
GET
END_GET
END_PROPERTY

{attribute 'TcRpcEnable'}
METHOD setOperation : BOOL
VAR_INPUT
	Operation	: AFE_CMD;
END_VAR
END_METHOD

{attribute 'monitoring' := 'call'}
{attribute 'TcRpcEnable'}
PROPERTY State : P6State
GET
END_GET
END_PROPERTY

END_INTERFACE

// NtoMProtocol/IProtoBaseNTo1
INTERFACE IProtoBaseNTo1 EXTENDS IProtoService

{attribute 'monitoring' := 'call'}
METHOD attach : IProtoBaseNTo1
VAR_INPUT
	Master	: IProtoMasterSingleService;
END_VAR
END_METHOD

{attribute 'monitoring' := 'call'}
METHOD getMasterByIdx : IProtoMasterSingleService
VAR_INPUT
	Index  : DINT;
END_VAR
END_METHOD

{attribute 'monitoring' := 'call'}
METHOD getNoMasters : DINT
END_METHOD

{attribute 'monitoring' := 'call'}
METHOD isAttached : BOOL
VAR_INPUT
	Master	: IProtoMasterSingleService;
END_VAR
END_METHOD

{attribute 'monitoring' := 'call'}
METHOD resetServices : IProtoBaseNTo1
END_METHOD

END_INTERFACE

// NtoMProtocol/IProtoMasterSingleService
INTERFACE IProtoMasterSingleService EXTENDS IProtocol

{attribute 'monitoring' := 'call'}
METHOD attach : IProtoMasterSingleService
VAR_INPUT
	Service	: IProtoService;
END_VAR
END_METHOD

{attribute 'monitoring' := 'call'}
METHOD getService : IProtoService
END_METHOD

END_INTERFACE

// Electrical/PMS/IPMS
INTERFACE IPMS

{attribute 'monitoring' := 'call'}
{attribute 'TcRpcEnable'}
METHOD attachAFE : IPMS
VAR_INPUT
	AFE : IProtoService;
END_VAR
END_METHOD

{attribute 'monitoring' := 'call'}
{attribute 'TcRpcEnable'}
METHOD attachInverter : IPMS
VAR_INPUT
	Inverter : IProtoService;
END_VAR
END_METHOD

{attribute 'monitoring' := 'call'}
{attribute 'TcRpcEnable'}
METHOD delAllAFE : IPMS
END_METHOD

{attribute 'monitoring' := 'call'}
{attribute 'TcRpcEnable'}
METHOD delAllInverters : IPMS
END_METHOD

{attribute 'monitoring' := 'call'}
{attribute 'TcRpcEnable'}
PROPERTY LimitPowerRegenUsage : BOOL
GET
END_GET
END_PROPERTY

{attribute 'monitoring' := 'call'}
{attribute 'TcRpcEnable'}
PROPERTY LimitPowerUsage : BOOL
GET
END_GET
END_PROPERTY

{attribute 'monitoring' := 'call'}
{attribute 'TcRpcEnable'}
PROPERTY PassiveMode : BOOL
GET
END_GET
SET
END_SET
END_PROPERTY

{attribute 'monitoring' := 'call'}
{attribute 'TcRpcEnable'}
PROPERTY PowerRegenUsage : LREAL
GET
END_GET
END_PROPERTY

{attribute 'monitoring' := 'call'}
{attribute 'TcRpcEnable'}
PROPERTY PowerUsage : LREAL
GET
END_GET
END_PROPERTY

{attribute 'monitoring' := 'call'}
{attribute 'TcRpcEnable'}
PROPERTY StopPowerUsage : BOOL
GET
END_GET
END_PROPERTY

END_INTERFACE

// Electrical/Softstarter/ISoftstarter
INTERFACE ISoftstarter

{attribute 'monitoring':='call'}
{attribute 'TcRpcEnable'}
PROPERTY Active : BOOL
GET
END_GET
SET
END_SET
END_PROPERTY

{attribute 'monitoring':='call'}
{attribute 'TcRpcEnable'}
PROPERTY Enabled : BOOL
GET
END_GET
SET
END_SET
END_PROPERTY

{attribute 'monitoring':='call'}
{attribute 'TcRpcEnable'}
PROPERTY Error : BOOL
GET
END_GET
END_PROPERTY

{attribute 'monitoring':='call'}
{attribute 'TcRpcEnable'}
PROPERTY Local : BOOL
GET
END_GET
END_PROPERTY

{attribute 'monitoring':='call'}
{attribute 'TcRpcEnable'}
PROPERTY OpTime : TIME
GET
END_GET
SET
END_SET
END_PROPERTY

{attribute 'monitoring':='call'}
{attribute 'TcRpcEnable'}
PROPERTY PowerUsage : LREAL
GET
END_GET
END_PROPERTY

(*
	This state bit is showing when the softstarter is ready to start a motor without a fault.  
*)
{attribute 'monitoring':='call'}
{attribute 'TcRpcEnable'}
PROPERTY Ready : BOOL
GET
END_GET
END_PROPERTY

{attribute 'TcRpcEnable'}
METHOD reset : BOOL
END_METHOD

{attribute 'monitoring':='call'}
{attribute 'TcRpcEnable'}
PROPERTY Running : BOOL
GET
END_GET
END_PROPERTY

{attribute 'TcRpcEnable'}
METHOD start : BOOL
END_METHOD

{attribute 'TcRpcEnable'}
METHOD stop : BOOL
END_METHOD

END_INTERFACE

// EStop/IEmergencyStop
INTERFACE IEmergencyStop

{attribute 'monitoring' := 'call'}
{attribute 'TcRpcEnable'}
PROPERTY Activated : BOOL
GET
END_GET
END_PROPERTY

{attribute 'monitoring' := 'call'}
{attribute 'TcRpcEnable'}
PROPERTY ActivatedSwitchIdx : INT
GET
END_GET
END_PROPERTY

{attribute 'monitoring' := 'call'}
{attribute 'TcRpcEnable'}
PROPERTY ActivatedSwitchName : P6IdName
GET
END_GET
END_PROPERTY

END_INTERFACE

// Hydraulics/HPU/IHPUBrake
INTERFACE IHPUBrake

{attribute 'monitoring' := 'call'}
{attribute 'TcRpcEnable'}
PROPERTY Active : BOOL
GET
END_GET
END_PROPERTY

{attribute 'monitoring' := 'call'}
{attribute 'TcRpcEnable'}
PROPERTY Error : BOOL
GET
END_GET
END_PROPERTY

{attribute 'monitoring' := 'call'}
{attribute 'TcRpcEnable'}
PROPERTY PressureOK : BOOL
GET
END_GET
END_PROPERTY

{attribute 'TcRpcEnable'}
METHOD setActive : BOOL
END_METHOD

END_INTERFACE

// Hydraulics/Valve/IValve
// Class to control a valve with solenoide 
INTERFACE IValve

{attribute 'monitoring' := 'call'}
{attribute 'TcRpcEnable'}
PROPERTY CalibrationMode : BOOL
GET
END_GET
END_PROPERTY

{attribute 'monitoring' := 'call'}
{attribute 'TcRpcEnable'}
PROPERTY Error : BOOL
GET
END_GET
END_PROPERTY

{attribute 'TcRpcEnable'}
METHOD setValve : BOOL
VAR_INPUT
	CMD		: ValveCMD;			// Command the valve output to be on or off
	value	: LREAL;			// Relative valve position. Range from 0-1 (0-100%).
END_VAR
END_METHOD

END_INTERFACE

// PID/IPID2DController
INTERFACE IPID2DController

{attribute 'TcRpcEnable'}
PROPERTY Error : LREAL
GET
END_GET
END_PROPERTY

{attribute 'TcRpcEnable'}
PROPERTY Out : LREAL
GET
END_GET
END_PROPERTY

{attribute 'TcRpcEnable'}
METHOD update : LREAL
VAR_INPUT
	config 				: REFERENCE TO ConfigPID2P;
	Active 				: BOOL;
	Setpoint 			: LREAL;
	ProcessValue 		: LREAL;
	ProcessValueFF1 	: LREAL;
	ProcessValueFF2 	: LREAL;	
	LowerBoundary 		: LREAL;
	UpperBoundary 		: LREAL;
	CycleTime			: LREAL;
END_VAR
END_METHOD

END_INTERFACE

// PID/IPIDController
INTERFACE IPIDController

{attribute 'TcRpcEnable'}
PROPERTY Error : LREAL
GET
END_GET
END_PROPERTY

{attribute 'TcRpcEnable'}
PROPERTY Out : LREAL
GET
END_GET
END_PROPERTY

{attribute 'TcRpcEnable'}
METHOD update : LREAL
VAR_INPUT
	config 				: REFERENCE TO ConfigPID;
	Active 				: BOOL;
	Setpoint 			: LREAL;
	ProcessValue 		: LREAL;
	ProcessValueFF1 	: LREAL;
	ProcessValueFF2 	: LREAL;	
	LowerBoundary 		: LREAL;
	UpperBoundary 		: LREAL;
	CycleTime			: LREAL;
END_VAR
END_METHOD

END_INTERFACE

// Sensor/IAnalogSensor
INTERFACE IAnalogSensor EXTENDS IAnalogSensorBase

{attribute 'monitoring' := 'call'}
{attribute 'TcRpcEnable'}
PROPERTY Error : BOOL
GET
END_GET
END_PROPERTY

END_INTERFACE

// Sensor/IAnalogSensorBase
INTERFACE IAnalogSensorBase EXTENDS __SYSTEM.IQueryInterface

{attribute 'monitoring' := 'call'}
{attribute 'TcRpcEnable'}
PROPERTY Value : LREAL
GET
END_GET
END_PROPERTY

{attribute 'monitoring' := 'call'}
{attribute 'TcRpcEnable'}
PROPERTY ValueRaw : LREAL
GET
END_GET
END_PROPERTY

END_INTERFACE

// Winch/IAnchorWinch
INTERFACE IAnchorWinch

END_INTERFACE

// Winch/IClutch
INTERFACE IClutch  EXTENDS __System.IQueryInterface

{attribute 'monitoring':='call'}
{attribute 'TcRpcEnable'}
PROPERTY ClutchState : ClutchStates
GET
END_GET
END_PROPERTY

// Set this TRUE to enable function
{attribute 'monitoring':='call'}
{attribute 'TcRpcEnable'}
PROPERTY ParkingBrakesOnWhileJoystickInCenterEnabled : BOOL
GET
END_GET
SET
END_SET
END_PROPERTY

{attribute 'TcRpcEnable'}
METHOD SetClutchOperation : BOOL
VAR_INPUT
	CMD : ClutchCMD;
END_VAR
END_METHOD

END_INTERFACE

// Winch/IClutchAndBrake
INTERFACE IClutchAndBrake  EXTENDS __System.IQueryInterface

//Brake pressure to be displayed.
{attribute 'monitoring':='call'}
{attribute 'TcRpcEnable'}
PROPERTY BrakeOffPressure : LREAL
GET
END_GET
END_PROPERTY

//Brake pressure to be displayed.
{attribute 'monitoring':='call'}
{attribute 'TcRpcEnable'}
PROPERTY BrakeOnPressure : LREAL
GET
END_GET
END_PROPERTY

{attribute 'monitoring':='call'}
{attribute 'TcRpcEnable'}
PROPERTY ClutchState : ClutchStates
GET
END_GET
END_PROPERTY

{attribute 'monitoring':='call'}
{attribute 'TcRpcEnable'}
PROPERTY FreeWheelingBrakeState : FreeWheelingBrakeStates
GET
END_GET
END_PROPERTY

// Set this TRUE to enable function
{attribute 'monitoring':='call'}
{attribute 'TcRpcEnable'}
PROPERTY ParkingBrakesOnWhileJoystickInCenterEnabled : BOOL
GET
END_GET
SET
END_SET
END_PROPERTY

{attribute 'TcRpcEnable'}
METHOD SetClutchOperation : BOOL
VAR_INPUT
	CMD : ClutchCMD;
END_VAR
END_METHOD

{attribute 'TcRpcEnable'}
METHOD SetFreeWheelingBrakeOperation : BOOL
VAR_INPUT
	CMD : FreeWheelingBrakeUserCMD;
END_VAR
END_METHOD

END_INTERFACE

// Winch/IFishpump
// Specialized user winch class to handle fishpump
INTERFACE IFishpump EXTENDS __SYSTEM.IQueryInterface

{attribute 'monitoring':='call'}
{attribute 'TcRpcEnable'}
PROPERTY DifferentialPressure : LREAL
GET
END_GET
END_PROPERTY

// Pressure outside fishpump
{attribute 'monitoring':='call'}
{attribute 'TcRpcEnable'}
PROPERTY EnvironmentalPressure : LREAL
GET
END_GET
END_PROPERTY

// Pressure inside motor housing
{attribute 'monitoring':='call'}
{attribute 'TcRpcEnable'}
PROPERTY MotorhousePressure : LREAL
GET
END_GET
END_PROPERTY

// Temperature of motor oil
{attribute 'monitoring':='call'}
{attribute 'TcRpcEnable'}
PROPERTY OilTemperature : LREAL
GET
END_GET
END_PROPERTY

{attribute 'monitoring':='call'}
{attribute 'TcRpcEnable'}
PROPERTY PressureLow : BOOL
GET
END_GET
END_PROPERTY

{attribute 'monitoring':='call'}
{attribute 'TcRpcEnable'}
PROPERTY TemperatureHigh : BOOL
GET
END_GET
END_PROPERTY

END_INTERFACE

// Winch/INetHaulerWinch
INTERFACE INetHaulerWinch

PROPERTY TiltIn : BOOL
SET
END_SET
END_PROPERTY

PROPERTY TiltOut : BOOL
SET
END_SET
END_PROPERTY

END_INTERFACE

// Winch/ISpool
INTERFACE ISpool EXTENDS IP6State, IP6OpState, __SYSTEM.IQueryInterface

{attribute 'TcRpcEnable'}
METHOD confirmWirePosition : BOOL
VAR_INPUT
END_VAR
END_METHOD

{attribute 'monitoring' := 'call'}
{attribute 'TcRpcEnable'}
PROPERTY HeadPosition : LREAL
GET
END_GET
END_PROPERTY

{attribute 'monitoring' := 'call'}
{attribute 'TcRpcEnable'}
PROPERTY Name : P6IdName
GET
END_GET
END_PROPERTY

{attribute 'monitoring' := 'call'}
{attribute 'TcRpcEnable'}
PROPERTY OpState : P6OpState
GET
END_GET
END_PROPERTY

{attribute 'monitoring' := 'call'}
{attribute 'TcRpcEnable'}
PROPERTY PIDError : LREAL
GET
END_GET
END_PROPERTY

{attribute 'TcRpcEnable'}
METHOD setManualOperation : BOOL
VAR_INPUT
	CMD : ManualSpoolCMD;
END_VAR
END_METHOD

{attribute 'TcRpcEnable'}
METHOD setOffsetDiamondScrew : BOOL
END_METHOD

{attribute 'TcRpcEnable'}
{attribute 'TcRpcEnable'}
METHOD setOperation : BOOL
VAR_INPUT
	CMD : SpoolCMD; 
END_VAR
END_METHOD

{attribute 'TcRpcEnable'}
METHOD setSpoolEndPositionInner : BOOL
VAR_INPUT
END_VAR
END_METHOD

{attribute 'TcRpcEnable'}
METHOD setSpoolEndPositionOuter : BOOL
VAR_INPUT
END_VAR
END_METHOD

{attribute 'monitoring' := 'call'}
{attribute 'TcRpcEnable'}
PROPERTY Speed : LREAL
GET
END_GET
END_PROPERTY

{attribute 'monitoring' := 'call'}
{attribute 'TcRpcEnable'}
PROPERTY State : P6State
GET
END_GET
END_PROPERTY

END_INTERFACE

// Winch/ITrawlModeController
INTERFACE ITrawlModeController EXTENDS IWinchMode, IP6OpState

// true if allowed to enter haul in modes. Both to setpoint and to safety range.
{attribute 'monitoring':='call'}
{attribute 'TcRpcEnable'}
PROPERTY HaulInModeAllowed : BOOL
GET
END_GET
END_PROPERTY

{attribute 'monitoring':='call'}
{attribute 'TcRpcEnable'}
PROPERTY LengthDifference : LREAL
GET
END_GET
END_PROPERTY

// The maximum allowed towing difference in auto trawl modes
{attribute 'monitoring':='call'}
{attribute 'TcRpcEnable'}
PROPERTY LengthDifferenceMax : LREAL
GET
END_GET
SET
END_SET
END_PROPERTY

// TRUE if difference in length between winches > MaxLengthDifference
{attribute 'monitoring':='call'}
{attribute 'TcRpcEnable'}
PROPERTY LengthDifferenceWarning : BOOL
GET
END_GET
END_PROPERTY

{attribute 'monitoring':='call'}
{attribute 'TcRpcEnable'}
PROPERTY LengthMaster : LREAL
GET
END_GET
END_PROPERTY

// The setpoint for length in auto trawl modes
{attribute 'monitoring':='call'}
{attribute 'TcRpcEnable'}
PROPERTY LengthSetpoint : LREAL
GET
END_GET
SET
END_SET
END_PROPERTY

// true if allowed to enter pay out mode.
{attribute 'monitoring':='call'}
{attribute 'TcRpcEnable'}
PROPERTY PayoutModeAllowed : BOOL
GET
END_GET
END_PROPERTY

// The safety length for trawl modes. Automodes are allowed outside safetyrange.
{attribute 'monitoring':='call'}
{attribute 'TcRpcEnable'}
PROPERTY SafetyLength : LREAL
GET
END_GET
SET
END_SET
END_PROPERTY

{attribute 'TcRpcEnable'}
METHOD setOperation : BOOL
VAR_INPUT
	Operation : TrawlWinchCMD;
END_VAR
END_METHOD

{attribute 'TcRpcEnable'}
METHOD setSounderDifferenceToZero : BOOL
END_METHOD

// Set this to true in HMI if TDE is enabled.
{attribute 'monitoring':='call'}
{attribute 'TcRpcEnable'}
PROPERTY SnagControl : BOOL
GET
END_GET
SET
END_SET
END_PROPERTY

//Gives out the difference in length between sounder and trawl winches 
{attribute 'monitoring':='call'}
{attribute 'TcRpcEnable'}
PROPERTY SounderLengthDifference : LREAL
GET
END_GET
END_PROPERTY

{attribute 'monitoring':='call'}
{attribute 'TcRpcEnable'}
PROPERTY SounderLengthDifferenceMax : LREAL
GET
END_GET
END_PROPERTY

{attribute 'monitoring':='call'}
{attribute 'TcRpcEnable'}
PROPERTY SounderLengthDifferenceWarning : BOOL
GET
END_GET
END_PROPERTY

// Set this to true in HMI if TDE is enabled.
{attribute 'monitoring':='call'}
{attribute 'TcRpcEnable'}
PROPERTY TDE : BOOL
GET
END_GET
SET
END_SET
END_PROPERTY

// true if allowed to enter towing mode.
{attribute 'monitoring':='call'}
{attribute 'TcRpcEnable'}
PROPERTY TowingModeAllowed : BOOL
GET
END_GET
END_PROPERTY

END_INTERFACE

// Winch/ITrawlWinch
INTERFACE ITrawlWinch EXTENDS IBaseUserWinch

{attribute 'monitoring' := 'call'}
{attribute 'TcRpcEnable'}
PROPERTY AutoAvailable : BOOL
GET
END_GET
END_PROPERTY

PROPERTY AutoMode : BOOL
GET
END_GET
SET
END_SET
END_PROPERTY

PROPERTY Radius : LREAL
GET
END_GET
END_PROPERTY

{attribute 'monitoring' := 'call'}
{attribute 'TcRpcEnable'}
PROPERTY SafetyDistance : LREAL
GET
END_GET
END_PROPERTY

{attribute 'monitoring':='call'}
{attribute 'TcRpcEnable'}
METHOD setOperation : BOOL
VAR_INPUT
	CMD : TrawlWinchCMD;
END_VAR
END_METHOD

PROPERTY TorqueAuto : LREAL
GET
END_GET
SET
END_SET
END_PROPERTY

PROPERTY VelocityAuto : LREAL
GET
END_GET
SET
END_SET
END_PROPERTY

END_INTERFACE
